TYPE T_SIM_SHUTTER_STAT :
STRUCT
	bInitialised:	BOOL	:= FALSE;						(* If TRUE, shutter simulator is initialised *)

	nErrorCode: 	DINT 	:= E_SHUTTER_ERROR.SIM_NOT_INITIALISED;	(* Error code *)
	sErrorText: 	STRING 	:= 'NOT INITIALISED'; 			(* Error text *)
	sStatus: 		STRING 	:= 'ERROR'; 					(* Shutter status in textual form, e.g. 'OFF' *)
END_STRUCT
END_TYPE

(* stored: Version 1.1.0.1, ProductVersion 3.1.4022.16
   DUT T_SIM_SHUTTER_STAT: Id {91af19d4-208f-48f7-a423-e4ef68fbafcd} *)
